TYPE Vec3d : ARRAY[1..3] OF LREAL; END_TYPE

(* stored: Version 1.1.0.1, ProductVersion 3.1.4024.12
   DUT Vec3d: Id {580f50cd-32df-4075-be65-645f14c4c841} *)
